FUNCTION_BLOCK Axis IMPLEMENTS itfAxis
VAR_INPUT
END_VAR
VAR_OUTPUT
END_VAR
VAR
END_VAR

{warning 'add method implementation '}
METHOD AccelerationProfile : itfCommand
VAR_INPUT
	TimeScale	: REAL;
	AccelerationScale	: REAL;
	Offset	: REAL;
	BufferMode	: MC_BUFFER_MODE;
END_VAR
END_METHOD

{warning 'add property implementation'}
PROPERTY ActualPosition : REAL
GET
END_GET
END_PROPERTY

{warning 'add property implementation'}
PROPERTY ActualTorque : REAL
GET
END_GET
END_PROPERTY

{warning 'add property implementation'}
PROPERTY ActualVelocity : REAL
GET
END_GET
END_PROPERTY

{warning 'add property implementation'}
PROPERTY AxisWarning : BOOL
GET
END_GET
END_PROPERTY

{warning 'add method implementation '}
METHOD CamIn : itfSynchronizedAxisCommand
VAR_INPUT
	Master	: itfAxis;
	MasterOffset	: REAL;
	SlaveOffset	: REAL;
	MasterScaling	: REAL;
	SlaveScaling	: REAL;
	MasterStartDistance	: REAL;
	MasterSyncPosition	: REAL;
	StartMode	: MC_StartMode;
	MasterValueSource	: MC_Source;
	CamTable	: itfCamTable;
	BufferMode	: MC_BUFFER_MODE;
END_VAR
END_METHOD

{warning 'add method implementation '}
METHOD CombineAxes : itfSynchronizedAxisCommand
VAR_INPUT
	Master1	: itfAxis;
	Master2	: itfAxis;
	CombineMode	: MC_COMBINE_MODE;
	GearRatioNumeratorM1	: INT;
	GearRatioDenominatorM1	: INT;
	GearRatioNumeratorM2	: INT;
	GearRatioDenominatorM2	: INT;
	MasterValueSourceM1	: MC_SOURCE;
	MasterValueSourceM2	: MC_SOURCE;
	BufferMode	: MC_BUFFER_MODE;
END_VAR
END_METHOD

{warning 'add property implementation'}
PROPERTY CommunicationReady : BOOL
GET
END_GET
END_PROPERTY

{warning 'add property implementation'}
PROPERTY Direction : AXIS_DIRECTION
GET
END_GET
END_PROPERTY

{warning 'add property implementation'}
PROPERTY ErrorId : WORD
GET
END_GET
END_PROPERTY

{warning 'add method implementation '}
METHOD GearIn : itfSynchronizedAxisCommand
VAR_INPUT
	Master	: itfAxis;
	Ratio	: REAL;
	MasterValueSource	: INT;
	Acceleration	: REAL;
	Deceleration	: REAL;
	Jerk	: REAL;
	BufferMode	: MC_BUFFER_MODE;
END_VAR
END_METHOD

{warning 'add method implementation '}
METHOD GearInPos : itfSynchronizedAxisCommand
VAR_INPUT
	Master	: itfAxis;
	RatioNumerator	: REAL;
	RatioDenominator	: REAL;
	MasterValueSource	: MC_SOURCE;
	MasterSyncPosition	: REAL;
	SlaveSyncPosition	: REAL;
	SyncMode	: MC_SYNC_MODE;
	MasterStartDistance	: REAL;
	Velocity	: REAL;
	Acceleration	: REAL;
	Deceleration	: REAL;
	Jerk	: REAL;
	BufferMode	: MC_BUFFER_MODE;
END_VAR
END_METHOD

{warning 'add method implementation '}
METHOD Halt : itfAxisCommand
VAR_INPUT
	Deceleration	: REAL;
	Jerk	: REAL;
	BufferMode	: MC_BUFFER_MODE;
END_VAR
END_METHOD

{warning 'add method implementation '}
METHOD HaltSuperimposed : itfAxisCommand
VAR_INPUT
	Deceleration	: REAL;
	Jerk	: REAL;
END_VAR
END_METHOD

{warning 'add method implementation '}
METHOD Home : itfAxisCommand
VAR_INPUT
	Position	: REAL;
	Velocity	: REAL;
	EndVelocity	: REAL;
	Acceleration	: REAL;
	Deceleration	: REAL;
	Jerk	: REAL;
	Direction	: MC_Direction;
	HomingMode	: INT;
	BufferMode	: MC_BUFFER_MODE;
END_VAR
END_METHOD

{warning 'add property implementation'}
PROPERTY HomeAbsSwitch : BOOL
GET
END_GET
END_PROPERTY

{warning 'add property implementation'}
PROPERTY IsHomed : BOOL
GET
END_GET
END_PROPERTY

{warning 'add property implementation'}
PROPERTY LimitSwitchNegative : BOOL
GET
END_GET
END_PROPERTY

{warning 'add property implementation'}
PROPERTY LimitSwitchPositive : BOOL
GET
END_GET
END_PROPERTY

{warning 'add property implementation'}
PROPERTY MotionStatus : MOTION_STATUS
GET
END_GET
END_PROPERTY

{warning 'add method implementation '}
METHOD MoveAbsolute : itfAxisCommand
VAR_INPUT
	Position	: REAL;
	Velocity	: REAL;
	Acceleration	: REAL;
	Deceleration	: REAL;
	Jerk	: REAL;
	Direction	: MC_Direction;
	BufferMode	: MC_BUFFER_MODE;
END_VAR
END_METHOD

{warning 'add method implementation '}
METHOD MoveAdditive : itfAxisCommand
VAR_INPUT
	Distance	: REAL;
	Velocity	: REAL;
	Acceleration	: REAL;
	Deceleration	: REAL;
	Jerk	: REAL;
	BufferMode	: MC_BUFFER_MODE;
END_VAR
END_METHOD

{warning 'add method implementation '}
METHOD MoveContinuousAbsolute : itfContinuousAxisCommand
VAR_INPUT
	Position	: REAL;
	EndVelocity	: REAL;
	Velocity	: REAL;
	Acceleration	: REAL;
	Deceleration	: REAL;
	Jerk	: REAL;
	Direction	: MC_DIRECTION;
	BufferMode	: MC_BUFFER_MODE;
END_VAR
END_METHOD

{warning 'add method implementation '}
METHOD MoveContinuousRelative : itfContinuousAxisCommand
VAR_INPUT
	Distance	: REAL;
	EndVelocity	: REAL;
	Velocity	: REAL;
	Acceleration	: REAL;
	Deceleration	: REAL;
	Jerk	: REAL;
	Direction	: MC_DIRECTION;
	BufferMode	: MC_BUFFER_MODE;
END_VAR
END_METHOD

{warning 'add method implementation '}
METHOD MoveRelative : itfAxisCommand
VAR_INPUT
	Distance	: REAL;
	Velocity	: REAL;
	Acceleration	: REAL;
	Deceleration	: REAL;
	Jerk	: REAL;
	BufferMode	: MC_BUFFER_MODE;
END_VAR
END_METHOD

{warning 'add method implementation '}
METHOD MoveSuperimposed : itfAxisCommand
VAR_INPUT
	Distance	: REAL;
	VelocityDiff	: REAL;
	Acceleration	: REAL;
	Deceleration	: REAL;
	Jerk	: REAL;
END_VAR
END_METHOD

{warning 'add method implementation '}
METHOD MoveVelocity : itfContinuousAxisCommand
VAR_INPUT
	Velocity	: REAL;
	Acceleration	: REAL;
	Deceleration	: REAL;
	Jerk	: REAL;
	Direction	: MC_Direction;
	BufferMode	: MC_BUFFER_MODE;
END_VAR
END_METHOD

{warning 'add method implementation '}
METHOD PhasingAbsolute : itfSynchronizedAxisCommand
VAR_INPUT
	Master	: itfAxis;
	PhaseShift	: REAL;
	Velocity	: REAL;
	Acceleration	: REAL;
	Deceleration	: REAL;
	Jerk	: REAL;
	BufferMode	: MC_BUFFER_MODE;
END_VAR
END_METHOD

{warning 'add method implementation '}
METHOD PhasingRelative : itfSynchronizedAxisCommand
VAR_INPUT
	Master	: itfAxis;
	PhaseShift	: REAL;
	Velocity	: REAL;
	Acceleration	: REAL;
	Deceleration	: REAL;
	Jerk	: REAL;
	BufferMode	: MC_BUFFER_MODE;
END_VAR
END_METHOD

{warning 'add method implementation '}
METHOD PositionProfile : itfCommand
VAR_INPUT
	TimeScale	: REAL;
	PositionScale	: REAL;
	Offset	: REAL;
	BufferMode	: MC_BUFFER_MODE;
END_VAR
END_METHOD

{warning 'add method implementation '}
METHOD Power : itfCommand
VAR_INPUT
	Enable	: BOOL;
	EnablePositive	: BOOL;
	EnableNegative	: BOOL;
END_VAR
END_METHOD

{warning 'add property implementation'}
PROPERTY PowerOn : BOOL
GET
END_GET
END_PROPERTY

{warning 'add method implementation '}
METHOD ReadBoolParameter : MC_Error
VAR_INPUT
	ParameterNumber	: INT;
END_VAR
VAR_OUTPUT
	Value	: BOOL;
END_VAR
END_METHOD

{warning 'add method implementation '}
METHOD ReadParameter : MC_Error
VAR_INPUT
	ParameterNumber	: INT;
END_VAR
VAR_OUTPUT
	Value	: REAL;
END_VAR
END_METHOD

{warning 'add property implementation'}
PROPERTY ReadyForPowerOn : BOOL
GET
END_GET
END_PROPERTY

{warning 'add method implementation '}
METHOD Release : MC_Error
END_METHOD

{warning 'add method implementation '}
METHOD Reset : itfCommand
END_METHOD

{warning 'add method implementation '}
METHOD SetOverride : MC_Error
VAR_INPUT
	VelFactor	: REAL;
	AccFactor	: REAL;
	JerkFactor	: REAL;
END_VAR
END_METHOD

{warning 'add method implementation '}
METHOD SetPosition : itfCommand
VAR_INPUT
	Position	: REAL;
	Relative	: BOOL;
	ExecutionMode	: MC_ExecutionMode;
END_VAR
END_METHOD

{warning 'add property implementation'}
PROPERTY Simulation : BOOL
GET
END_GET
END_PROPERTY

{warning 'add property implementation'}
PROPERTY Status : AXIS_STATUS
GET
END_GET
END_PROPERTY

{warning 'add method implementation '}
METHOD Stop : itfAxisCommand
VAR_INPUT
	Deceleration	: REAL;
	Jerk	: REAL;
END_VAR
END_METHOD

{warning 'add method implementation '}
METHOD TorqueControl : itfAxisCommand
VAR_INPUT
	Torque	: REAL;
	TorqueRamp	: REAL;
	Velocity	: REAL;
	Acceleration	: REAL;
	Deceleration	: REAL;
	Jerk	: REAL;
	Direction	: MC_DIRECTION;
	BufferMode	: MC_BUFFER_MODE;
END_VAR
END_METHOD

{warning 'add method implementation '}
METHOD VelocityProfile : itfCommand
VAR_INPUT
	TimeScale	: REAL;
	VelocityScale	: REAL;
	Offset	: REAL;
	BufferMode	: MC_BUFFER_MODE;
END_VAR
END_METHOD

{warning 'add method implementation '}
METHOD WriteBoolParameter : MC_Error
VAR_INPUT
	ParameterNumber	: INT;
	Value	: BOOL;
END_VAR
END_METHOD

{warning 'add method implementation '}
METHOD WriteParameter : MC_Error
VAR_INPUT
	ParameterNumber	: INT;
	Value	: REAL;
END_VAR
END_METHOD

END_FUNCTION_BLOCK

(* stored: Version 1.1.0.1, ProductVersion 3.1.4024.12
   POU Axis: Id {a2da1341-2a89-43f6-a974-acbc9590e668}, SpecialFunc None
   Method AccelerationProfile: Id {9c672153-ada2-4cdc-bbe2-6e6d7c238259}
   Property ActualPosition: Id {afa4713c-09aa-4997-90cf-97c737902a7f}
   Get Get: Id {953b0b1f-0252-4613-b62e-e68642f2eee1}
   Property ActualTorque: Id {e002586c-4f91-4864-b611-c03ae675b5e6}
   Get Get: Id {9f30c7ff-23dd-4c6d-9fcd-5276ab3664a9}
   Property ActualVelocity: Id {81f1d51e-e9c5-4a77-88e1-eab6e2e32d59}
   Get Get: Id {810ed4ab-a9e3-4f07-90df-607cb5c74797}
   Property AxisWarning: Id {78f5c2a0-5328-4781-9c41-703776f815a1}
   Get Get: Id {be9c54ef-15b0-461d-92da-329ca8f69788}
   Method CamIn: Id {efd9f51d-d2cc-41c3-8963-774719124bbb}
   Method CombineAxes: Id {4c4de45a-08b0-4331-965e-243e508687b7}
   Property CommunicationReady: Id {a3d2b117-c407-44fa-a8c1-d2eff9d3ba44}
   Get Get: Id {48f743db-684d-4b17-826d-5c512bf874f3}
   Property Direction: Id {9cf6eac8-7564-4362-985e-df70f59390d1}
   Get Get: Id {85f1b1ef-a4fe-479a-b7d1-1077d40c6e2d}
   Property ErrorId: Id {e499a203-6c0a-4599-9c06-ae67747a7395}
   Get Get: Id {89d6c0ec-e9d3-4283-9e46-cc10df42c6a7}
   Method GearIn: Id {275d50ef-fbd7-4b8c-bb80-0fdbf59ba4db}
   Method GearInPos: Id {3325f679-2ef1-4c58-bfb1-c069b6c6ede0}
   Method Halt: Id {d42eee94-3339-413e-9247-7f58f41e468e}
   Method HaltSuperimposed: Id {0201181c-8fe9-4a36-b35a-832f8a020dd5}
   Method Home: Id {44a4f845-bbe5-4ee4-af7b-19d29c5783fd}
   Property HomeAbsSwitch: Id {5a63b7df-b436-4dbc-8a04-0c557a4e7fd5}
   Get Get: Id {8c2487cd-4874-405d-9c6a-4d9bb0fc6e22}
   Property IsHomed: Id {5ba5bbfd-4dc5-4ec4-9649-c5fd3ccf5c78}
   Get Get: Id {c01e975c-d3d1-49d0-819d-8aec63178674}
   Property LimitSwitchNegative: Id {2573064e-0307-4b95-8799-bcd62b0d3255}
   Get Get: Id {740a4b1a-240b-4339-af1d-c497a57de78a}
   Property LimitSwitchPositive: Id {d55cddfb-01ee-4be5-a78c-3cbb19538926}
   Get Get: Id {d384304b-c609-4424-8713-97fdc7644ce5}
   Property MotionStatus: Id {d84d6d10-2dcf-4e74-ba10-e415ffd01394}
   Get Get: Id {57e778fd-cae1-4b6f-88a0-203bc52c60ae}
   Method MoveAbsolute: Id {93e717f8-47ab-4727-b1f6-0d6cd6144fda}
   Method MoveAdditive: Id {289ad395-b2f3-4703-bfc4-ce76dab666da}
   Method MoveContinuousAbsolute: Id {4f9d7f8d-23dc-4404-ba45-cd8cbe2ee3b4}
   Method MoveContinuousRelative: Id {85f6c482-72ff-45be-8d3c-e60cb64ff872}
   Method MoveRelative: Id {2034c9d9-ba0a-450f-8eaf-7dda8aa9fe7f}
   Method MoveSuperimposed: Id {4e3f05aa-ad13-4531-a70a-235858c4002e}
   Method MoveVelocity: Id {1a8e8b56-3128-4bfd-813a-6c486ace495e}
   Method PhasingAbsolute: Id {f701a397-8423-44fb-b443-b9f01efa3a5e}
   Method PhasingRelative: Id {669a88c7-4a7b-4fd9-a78f-b903869754c3}
   Method PositionProfile: Id {e4750493-0209-4ef9-b064-1884b2d57dc3}
   Method Power: Id {3b07a63d-c32b-4cb3-9018-50a820bd5fb0}
   Property PowerOn: Id {574e2c8a-0eac-439f-90f7-51d8c7d06448}
   Get Get: Id {b11d4181-e1dc-4afd-9f1e-c163135fd68b}
   Method ReadBoolParameter: Id {a02162a1-1836-4460-a687-b7bd729ad2c4}
   Method ReadParameter: Id {3a6308e1-9724-4218-adc8-88ce0d24bbc6}
   Property ReadyForPowerOn: Id {af2191da-a1fd-4b87-8749-7e5f8c668cb9}
   Get Get: Id {dd395027-2ed8-4eee-a4f5-f4aef3e1b638}
   Method Release: Id {3fdbdf61-7535-4fb9-9081-e17a82d585ee}
   Method Reset: Id {6f309915-04d4-4cf6-9722-63a53f82afae}
   Method SetOverride: Id {82a8e42a-06d2-42e9-8c65-846187503543}
   Method SetPosition: Id {b9ab4cf6-8988-41ef-9bb2-0b01d3acc6f5}
   Property Simulation: Id {9448b4db-5b42-41b4-a743-358b5f52ef73}
   Get Get: Id {7fdb09f8-a103-4827-bc73-ecafaef03e0d}
   Property Status: Id {173a581e-a0c8-4747-88e9-ff58f6cf9216}
   Get Get: Id {afa65e67-d9ee-45e5-9980-2353f617b894}
   Method Stop: Id {483709e2-d443-4fe4-9c5f-7b1179b37ef6}
   Method TorqueControl: Id {88347a4e-d17b-49fc-855f-9fc006b85895}
   Method VelocityProfile: Id {51fd23ee-6a06-4ade-8a64-4f3726500273}
   Method WriteBoolParameter: Id {717080af-30a8-47ad-8ec3-340a3297b3d7}
   Method WriteParameter: Id {ceeedcb2-d45b-457e-9211-285d71fee8bb} *)
